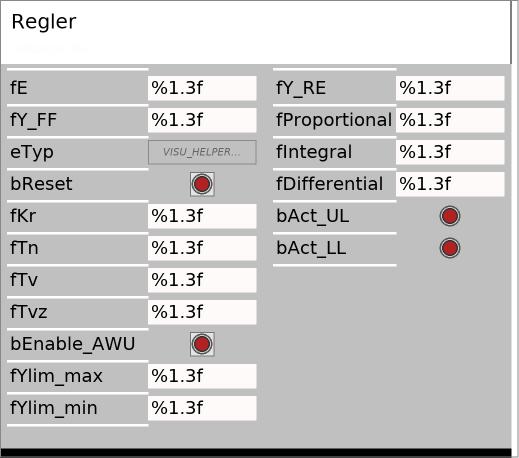
VISUALIZATION RET_VISU_Regler  // 519x458
VAR_INPUT
   {attribute 'parameterstringof' := 'm_Input_FB'}
   m_Input_INST_Str : STRING;
END_VAR
VAR_IN_OUT
   m_Input_FB : Regler;
END_VAR
    RoundedRectangle (0,0 511x81)
    RoundedRectangle (0,418 511x40)
    Rectangle (0,64 511x384)
    Lamp1 (438,204 24x24), variable: m_Input_FB.bAct_UL, style: Lamp-Lamp1-Red
    Lamp1 (438,236 24x24), variable: m_Input_FB.bAct_LL, style: Lamp-Lamp1-Red
    PushSwitch (190,172 24x24), variable: m_Input_FB.bReset, behaviour: TOGGLE, style: Switch-PushSwitch-Red
    PushSwitch (190,332 24x24), variable: m_Input_FB.bEnable_AWU, behaviour: TOGGLE, style: Switch-PushSwitch-Red
    Rectangle (8,8 511x27), "Regler"
    Rectangle (8,35 511x27), "Instance: %s", text variable: m_Input_INST_Str
    Rectangle (7,68 141x2)
    Rectangle (148,76 108x24), "%1.3f", text variable: m_Input_FB.fE
        OnMouseClick: write the text variable via Default
    Rectangle (7,76 141x24), "fE"
    Rectangle (7,104 141x2)
    Rectangle (148,108 108x24), "%1.3f", text variable: m_Input_FB.fY_FF
        OnMouseClick: write the text variable via Default
    Rectangle (7,108 141x24), "fY_FF"
    Rectangle (7,136 141x2)
    Rectangle (7,140 141x24), "eTyp"
    Rectangle (7,168 141x2)
    Rectangle (7,172 141x24), "bReset"
    Rectangle (7,200 141x2)
    Rectangle (148,204 108x24), "%1.3f", text variable: m_Input_FB.fKr
        OnMouseClick: write the text variable via Default
    Rectangle (7,204 141x24), "fKr"
    Rectangle (7,232 141x2)
    Rectangle (148,236 108x24), "%1.3f", text variable: m_Input_FB.fTn
        OnMouseClick: write the text variable via Default
    Rectangle (7,236 141x24), "fTn"
    Rectangle (7,264 141x2)
    Rectangle (148,268 108x24), "%1.3f", text variable: m_Input_FB.fTv
        OnMouseClick: write the text variable via Default
    Rectangle (7,268 141x24), "fTv"
    Rectangle (7,296 141x2)
    Rectangle (148,300 108x24), "%1.3f", text variable: m_Input_FB.fTvz
        OnMouseClick: write the text variable via Default
    Rectangle (7,300 141x24), "fTvz"
    Rectangle (7,328 141x2)
    Rectangle (7,332 141x24), "bEnable_AWU"
    Rectangle (7,360 141x2)
    Rectangle (148,364 108x24), "%1.3f", text variable: m_Input_FB.fYlim_max
        OnMouseClick: write the text variable via Default
    Rectangle (7,364 141x24), "fYlim_max"
    Rectangle (7,392 141x2)
    Rectangle (148,396 108x24), "%1.3f", text variable: m_Input_FB.fYlim_min
        OnMouseClick: write the text variable via Default
    Rectangle (7,396 141x24), "fYlim_min"
    Rectangle (7,424 141x2)
    Rectangle (273,68 123x2)
    Rectangle (396,76 108x24), "%1.3f", text variable: m_Input_FB.fY_RE
    Rectangle (273,76 123x24), "fY_RE"
    Rectangle (273,104 123x2)
    Rectangle (396,108 108x24), "%1.3f", text variable: m_Input_FB.fProportional
    Rectangle (273,108 123x24), "fProportional"
    Rectangle (273,136 123x2)
    Rectangle (396,140 108x24), "%1.3f", text variable: m_Input_FB.fIntegral
    Rectangle (273,140 123x24), "fIntegral"
    Rectangle (273,168 123x2)
    Rectangle (396,172 108x24), "%1.3f", text variable: m_Input_FB.fDifferential
    Rectangle (273,172 123x24), "fDifferential"
    Rectangle (273,200 123x2)
    Rectangle (273,204 123x24), "bAct_UL"
    Rectangle (273,232 123x2)
    Rectangle (273,236 123x24), "bAct_LL"
    Rectangle (273,264 123x2)
    Frame (148,140 108x24), input disabled if: False
        shows VISU_HELPER_Combobox_eReglertyp(varEnum := m_Input_FB.eTyp)
END_VISUALIZATION

(* stored: Version 1.1.0.1, ProductVersion 3.1.4024.12
   Visu RET_VISU_Regler: Id {13b3ea54-bec2-4493-b2f9-57d22bd5cb4f} *)
